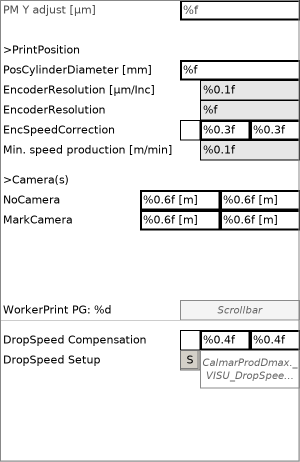
VISUALIZATION _VISU_Pm_Settings  // 300x462
VAR_IN_OUT
	mInst : FB_PrintModule_WEU;
END_VAR
    Rectangle (0,60 180x20), "PosCylinderDiameter [mm]"
    Rectangle (0,80 180x20), "EncoderResolution [µm/Inc]"
    Rectangle (200,80 100x20), "%0.1f", tooltip "constant", text variable: mInst.fC_EncoderImpU
    Rectangle (180,60 120x20), "%f", text variable: mInst._fEncoderCylinderDiameter
        OnMouseClick: write the text variable via Default
    Rectangle (0,0 180x20), "PM Y adjust [µm]"
    Rectangle (180,0 120x20), "%f", text variable: mInst._fPrintModuleAdjustY
        OnMouseClick: write the text variable via VisuDialogs.Numpad, min PRG_PRINT.sC_Config_P.lL_PU_GENERALSHIFT_Y_SET_MIN, max PRG_PRINT.sC_Config_P.lL_PU_GENERALSHIFT_Y_SET_MAX
    Rectangle (250,120 50x20), "%0.3f", tooltip "Encoder speed compensation reference speed", text variable: mInst.fbPrintPosition._fSpeedCompRefSpeed
        OnMouseClick: write the text variable via Default
    Rectangle (200,120 50x20), "%0.3f", tooltip "Encoder speed compensation factor", text variable: mInst.fbPrintPosition._fSpeedCompFactor
        OnMouseClick: write the text variable via Default
    RoundedRectangle (180,120 20x20)
        toggle mInst.fbPrintPosition._bEnSpeedComp
    Rectangle (0,120 180x20), "EncSpeedCorrection"
    Rectangle (0,100 180x20), "EncoderResolution"
    Rectangle (200,100 100x20), "%f", tooltip "by calculation", text variable: mInst.fbPrintPosition._fEncoderResolution
    Scrollbar (180,300 120x20)
        p2245068023: GVL_WEU.nC_WorkerPrintPerPm
        p1057716461: mInst.fbView.nSelWorkerPrint
    Rectangle (0,300 160x20), "WorkerPrint PG: %d", text variable: mInst.fbView.nSelWorkerPrint
    Rectangle (0,320 300x142)
    Rectangle (0,330 180x20), "DropSpeed Compensation"
    Rectangle (200,330 50x20), "%0.4f", tooltip "DropSpeed [m/s]", text variable: mInst.fbWorkerPrint[mInst.fbView.nSelWorkerPrint].fbDropSpeedComp.fDropSpeed
        OnMouseClick: write the text variable via Default
    Rectangle (250,330 50x20), "%0.4f", tooltip "Dead/Add Time [ms]", text variable: mInst.fbWorkerPrint[mInst.fbView.nSelWorkerPrint].fbDropSpeedComp.fDropSpeedDeadTime
        OnMouseClick: write the text variable via Default
    RoundedRectangle (180,330 20x20), tooltip "Enabled compensation", input disabled if: TRUE
        toggle mInst.fbWorkerPrint[mInst.fbView.nSelWorkerPrint].fbDropSpeedComp._bEnable p2164770859=TRUE
    Button (180,350 20x20), "S", tooltip "Setup"
        toggle minst.fbView.bShowDropSpeedSetup
    Rectangle (0,350 180x20), "DropSpeed Setup"
    Frame (200,350 100x38), invisible if: NOT minst.fbView.bShowDropSpeedSetup
        shows CalmarProdDmax._VISU_DropSpeedComp_Setup(mInst := mInst.fbWorkerPrint[mInst.fbView.nSelWorkerPrint].fbDropSpeedComp)
    Rectangle (0,40 180x20), ">PrintPosition"
    Rectangle (0,140 180x20), "Min. speed production [m/min]"
    Rectangle (200,140 100x20), "%0.1f", tooltip "constant", text variable: mInst.fC_ProductionSpeedMpMin_Level
    Rectangle (0,170 180x20), ">Camera(s)"
    Rectangle (220,190 80x20), "%0.6f [m]", tooltip "CameraToPrintUnit", text variable: mInst.fbNoCamera._fCameraToPrintOffset
        OnMouseDown: write the text variable via Default
    Rectangle (140,190 80x20), "%0.6f [m]", tooltip "DetectToCamera", text variable: mInst.fbNoCamera._fDetectToCameraOffset
        OnMouseDown: write the text variable via Default
    Rectangle (0,190 140x20), "NoCamera"
    Rectangle (220,210 80x20), "%0.6f [m]", tooltip "CameraToPrintUnit", text variable: mInst.fbMarkCameraWeu._fCameraToPrintOffset
        OnMouseDown: write the text variable via Default
    Rectangle (140,210 80x20), "%0.6f [m]", tooltip "DetectToCamera", text variable: mInst.fbMarkCameraWeu._fDetectToCameraOffset
        OnMouseDown: write the text variable via Default
    Rectangle (0,210 140x20), "MarkCamera"
END_VISUALIZATION

(* stored: Version 1.1.0.1, ProductVersion 3.1.4024.11
   Visu _VISU_Pm_Settings: Id {437752a8-825f-4ae5-b356-49b664924b0e} *)
